// TIA Portal V20 export
ORGANIZATION_BLOCK "Main"   // OB1, LAD, ProgramCycle
TITLE = "Main Program Sweep (Cycle)"
{ S7_Optimized_Access := 'TRUE' }
// stored: SetENOAutomatically false
   VAR_INPUT
      Initial_Call : Bool;   // Initial call of this OB
      Remanence : Bool;   // =True, if remanent data are available
   END_VAR
   VAR_TEMP   // added for the SCL form of the ladder/FBD networks
      _w1 : Bool;
   END_VAR
BEGIN

REGION Network 1
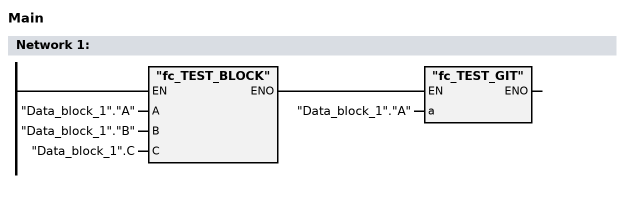
   RUNG wire#powerrail
      "fc_TEST_BLOCK"("A" := "Data_block_1"."A", "B" := "Data_block_1"."B", C := "Data_block_1".C)
      "fc_TEST_GIT"("a" := "Data_block_1"."A")
   END_RUNG
   // the same network as SCL:
   "fc_TEST_BLOCK"("A" := "Data_block_1"."A", "B" := "Data_block_1"."B", C := "Data_block_1".C, ENO => #_w1);
   IF #_w1 THEN "fc_TEST_GIT"("a" := "Data_block_1"."A"); END_IF;
END_REGION
END_ORGANIZATION_BLOCK
